(* CODESYS project Estação 3 - separating V2 (2022).project

Project tree, tasks and I/O mapping:
  Device : CPX-CEC-C1-V3, Festo AG & Co. KG, order no. 3473128, version 3.5.7.37
      unmapped channels: Rotary switch
    application Application
      libraries: Standard, * (System)
      task MainTask (cyclic, interval t#20ms, priority 20) calls PLC_PRG
      program PLC_PRG [ST]
      global variables GVL
      function ATUALIZAR_VALORES [ST]
      program pisca_pisca [ST]
      program modo_entrada [ST]
      program modo_saida [ST]
      program teste_comunicacao [ST]
    PLC_Diagnosis : PLC-Diagnosis, Festo AG & Co. KG, version 3.5.4.1
    CPX_System : CPX_System, Festo AG & Co. KG, order no. 3473128, version 1.258
      CEC_C1_V3 : CEC-C1-V3, Festo AG & Co. KG, order no. 3473128, version 1.258
          settings:  = 0;  = 234279157108224;  = 335718592;  = 65535;  = 16885952;  = 13959208;  = 1f5d13d5;  = 5
      _8DI_8DO : 8DI/8DO, Festo AG & Co. KG, order no. 526257, version 1.258
          settings:  = 0;  = 1;  = 1;  = 1;  = 1;  = 0;  = 1;  = 1;  = 0;  = 0;  = 0;  = 0;  = 0;  = 0;  = 0;  = 0;  = 0;  = 0;  = 0;  = 0;  = 0;  = 0;  = 0;  = 0;  = 0;  = 0;  = 0;  = 0;  = 0;  = 0;  = 0;  = 0;  = 0;  = 0;  = 0;  = 0;  = 0;  = 0;  = 0;  = 0;
             = 0;  = 0;  = 0;  = 0;  = 0;  = 0;  = 0;  = 0;  = 0;  = 0;  = 0;  = 0;  = 0;  = 0;  = 0;  = 0;  = 0;  = 0;  = 0;  = 0;  = 0;  = 0;  = 0;  = 0;  = 0;  = 0;  = 0;  = 0;  = 0;  = 0;  = 0;  = 0;  = 0;  = 0;  = 0;  = 0;  = 0;  = 0;  = 0;  = 0;
             = 576751027668385792;  = 'PI%i.0.0.1=1';  = 'PI%i.0.1.1=1';  = 'PI%i.0.2.1=1';  = 'PI%i.1.0.1=1';  = 'PI%i.1.1.1=0';  = 'PI%i.1.4.2=1';  = 'PI%i.1.6.2=1';  = 'PI%i.6.0.1=0';  = 'PI%i.6.1.1=0';  = 'PI%i.6.2.1=0';  = 'PI%i.6.3.1=0';  = 'PI%i.6.4.1=0';  = 'PI%i.6.5.1=0';  = 'PI%i.6.6.1=0';  = 'PI%i.6.7.1=0';  = dd379be8;  = 6
          unmapped channels: Input 0, Output 0
      _8DI_8DO_1 : 8DI/8DO, Festo AG & Co. KG, order no. 526257, version 1.258
          settings:  = 0;  = 1;  = 1;  = 1;  = 1;  = 0;  = 1;  = 1;  = 0;  = 0;  = 0;  = 0;  = 0;  = 0;  = 0;  = 0;  = 0;  = 0;  = 0;  = 0;  = 0;  = 0;  = 0;  = 0;  = 0;  = 0;  = 0;  = 0;  = 0;  = 0;  = 0;  = 0;  = 0;  = 0;  = 0;  = 0;  = 0;  = 0;  = 0;  = 0;
             = 0;  = 0;  = 0;  = 0;  = 0;  = 0;  = 0;  = 0;  = 0;  = 0;  = 0;  = 0;  = 0;  = 0;  = 0;  = 0;  = 0;  = 0;  = 0;  = 0;  = 0;  = 0;  = 0;  = 0;  = 0;  = 0;  = 0;  = 0;  = 0;  = 0;  = 0;  = 0;  = 0;  = 0;  = 0;  = 0;  = 0;  = 0;  = 0;  = 0;
             = 576751027668385792;  = 'PI%i.0.0.1=1';  = 'PI%i.0.1.1=1';  = 'PI%i.0.2.1=1';  = 'PI%i.1.0.1=1';  = 'PI%i.1.1.1=0';  = 'PI%i.1.4.2=1';  = 'PI%i.1.6.2=1';  = 'PI%i.6.0.1=0';  = 'PI%i.6.1.1=0';  = 'PI%i.6.2.1=0';  = 'PI%i.6.3.1=0';  = 'PI%i.6.4.1=0';  = 'PI%i.6.5.1=0';  = 'PI%i.6.6.1=0';  = 'PI%i.6.7.1=0';  = dd4a6df2;  = 6
          unmapped channels: Input 0, Output 0
    Ethernet : Ethernet, 3S - Smart Software Solutions GmbH, version 3.5.10.0
        settings: IPAddress = [192,168,0,1]; SubnetMask = [255,255,255,0]; GatewayAddress = [0,0,0,0]; MACAddress = [16#00,16#00,16#00,16#00,16#00,16#00]; SaveCommunicationSettings = FALSE
      ModbusTCP_Slave_Device : ModbusTCP Slave Device, 3S - Smart Software Solutions GmbH, version 3.5.10.0
          unmapped channels: Inputs, Outputs
*)

// Device/Application/GVL
	
{attribute 'qualified_only'}
VAR_GLOBAL
//Entradas
	//Sensores
	S_inicio 	AT %IX1.0 :BOOL; //Sensor de inicio da esteira
	S_meio 	 	AT %IX1.1 :BOOL; //Sensor do meio da esteira
	S_fim 		AT %IX1.2 :BOOL; //Sensor do fim da esteira
	S_dist		AT %IX1.3 :BOOL; //Sensor de distancia (sinal digital)
	S_inicio_2 	AT %IX1.4  :BOOL; //Sensor de inicio da esteira 2
	//  	AT %IX1.5  :BOOL; //
	S_fim_2 	AT %IX1.6  :BOOL; //Sensor do fim da esteira 2
	
	
	//IHM
	Start_btn 		AT	%IX2.0	:BOOL;  //Botão de start
	Stop_btn 		AT	%IX2.1	:BOOL;	//Botão de stop (NF)
	Chave 			AT	%IX2.2	:BOOL;	//Chave auto/manual
	Reset_btn 		AT	%IX2.3	:BOOL;	//Botão de reset
	I4_IHM			AT	%IX2.4	:BOOL;	//Bit de saída 4 da IHM
	I5_IHM			AT	%IX2.5	:BOOL;	//Bit de saída 5 da IHM
	I6_IHM 			AT	%IX2.6	:BOOL;	//Bit de saída 6 da IHM
	I7_IHM			AT	%IX2.7	:BOOL;	//Bit de saída 7 da IHM

//Saídas
	//Atuadorres 			
	Esteira_frente 	AT	%QX0.0	:BOOL;	//Mover a esteira 1 para frente
	Esteira_tras 	AT	%QX0.1	:BOOL;	//Mover a esteira 1 para tras
	Separador 	 	AT	%QX0.2	:BOOL;	//Atuar separador
	Stopper		 	AT	%QX0.3	:BOOL;	//Avança stopper
	Esteira_frente_2 AT	%QX0.4	:BOOL;	//Mover a esteira 2 para frente
	Esteira_tras_2	 AT	%QX0.5	:BOOL;	//Mover a esteira 2 para tras
	//				AT	%QX0.6	:BOOL;	
	//	     		AT	%QX0.7	:BOOL;	
	
	//IHM				
	Start_LED		AT	%QX1.0	:BOOL;	//LED do botão de start
	Reset_LED 		AT	%QX1.1	:BOOL;	//LED do botão de reset
	Q1_LED 			AT	%QX1.2	:BOOL;	//LED sinalizador Q1
	Q2_LED			AT	%QX1.3	:BOOL;	//LED sinalizador Q2
	Q4_IHM			AT	%QX1.4	:BOOL;	//Saída Q4 IHM
	Q5_IHM			AT	%QX1.5	:BOOL;	//Saída Q5 IHM
	Q6_IHM			AT	%QX1.6	:BOOL;	//Saída Q6 IHM
	Q7_IHM 			AT	%QX1.7	:BOOL;	//Saída Q7 IHM
	
//MODBUS bits
	//Entradas
	Mod_I_0_0 		AT %IX4.0 : BOOL; //Iniciar a estação 
	Mod_I_0_1	 	AT %IX4.1 : BOOL; //Parar a estação
	Mod_I_0_2 		AT %IX4.2 : BOOL; //Reiniciar a estação
	Mod_I_0_3 		AT %IX4.3 : BOOL; //Modo entrada
	Mod_I_0_4 		AT %IX4.4 : BOOL; ///Modo saída
	Mod_I_0_5 		AT %IX4.5 : BOOL; //Teste de resposta da estação - IN
	Mod_I_0_6 		AT %IX4.6 : BOOL;
	Mod_I_0_7 		AT %IX4.7 : BOOL;
	Mod_I_1_0 		AT %IX5.0 : BOOL;
	Mod_I_1_1 		AT %IX5.1 : BOOL;
	Mod_I_1_2 		AT %IX5.2 : BOOL;
	Mod_I_1_3 		AT %IX5.3 : BOOL;
	Mod_I_1_4 		AT %IX5.4 : BOOL;
	Mod_I_1_5	 	AT %IX5.5 : BOOL;
	Mod_I_1_6 		AT %IX5.6 : BOOL;
	Mod_I_1_7 		AT %IX5.7 : BOOL;
	
	//Saídas
	Mod_Q_0_0 		AT %QX2.0 : BOOL; //Estação iniciada 					
	Mod_Q_0_1	 	AT %QX2.1 : BOOL; //Estação parada 					
	Mod_Q_0_2 		AT %QX2.2 : BOOL; //Estação em processo			
	Mod_Q_0_3 		AT %QX2.3 : BOOL; //Estação em modo de entrada
	Mod_Q_0_4 		AT %QX2.4 : BOOL; //Estação em modo de saída
	Mod_Q_0_5 		AT %QX2.5 : BOOL; //Teste de resposta da estação - OUT	


//Variáveis de lógica
	principal: BOOL;
	parada : BOOL;
	passo1: BOOL;	
	passo2: BOOL;
	passo3: BOOL;
	passo4: BOOL;
	passo5: BOOL;
	passo6: BOOL;
	passo7: BOOL;
	passo8: BOOL;
	
	start: BOOL; //Start geral
	stop: BOOL;  //Stop geral
	reset: BOOL; //Reset geral
	key: BOOL; //key geral
	
	estacao_iniciada:  BOOL; //Flag para sinalizar que a estação está iniciada e pode receber algum comando
	estacao_parada: BOOL;	//Flag que sinaliza estação parada
	estacao_em_processo: BOOL; //Flag que sinaliza a estação em processo
	ligar_pisca: BOOL := FALSE; //Flag para ligar e desligar o pisca pisca
	modo_entrada: BOOL; //Quando setado, a estação entra em modo de saída de peças
	modo_saida: BOOL; //Quando setado, a estação entra em modo de entrada de peças
	Peca_robo: BOOL; //Quando for TRUE, a peça irá para a montagem no robô, se for FALSE irá para a montatgem da tampinha

END_VAR

// Device/Application/PLC_PRG
PROGRAM PLC_PRG
VAR
	TONInst4: Ton;
	TON_4: BOOL;
	TON_3: BOOL;
	TONInst3: Ton;
	TONInst1: Ton;
	TON_1: BOOL;
	TONInst2: Ton;
	TON_2: BOOL;
	TONInst5: Ton;
	TON_5: BOOL;
END_VAR

modo_entrada();
modo_saida();
pisca_pisca();
teste_comunicacao();
ATUALIZAR_VALORES();

END_PROGRAM

// Device/Application/modo_entrada
PROGRAM modo_entrada
VAR

	TON_temp_1: TON;
	TON_1: BOOL;
	
	TON_temp_2: TON;
	TON_2: BOOL;	
	
	PASSOS: INT;
	
END_VAR

TON_temp_1(IN := TON_1, PT:= T#0.5S);
TON_temp_2(IN := TON_2, PT:= T#0.4S);

IF NOT gvl.estacao_parada AND gvl.estacao_iniciada THEN
	
	IF (gvl.modo_entrada AND NOT gvl.modo_saida AND PASSOS = 0) THEN
		GVL.Q4_IHM := TRUE;
	END_IF
	
	IF ((gvl.modo_entrada AND NOT gvl.modo_saida) OR PASSOS = 1) AND gvl.S_inicio THEN
		GVL.Q4_IHM := FALSE;
		gvl.ligar_pisca := TRUE;
		gvl.estacao_em_processo := TRUE;
		gvl.Stopper := FALSE;	
		gvl.Esteira_frente := TRUE;
		gvl.Esteira_frente_2 := TRUE;
		gvl.Separador := TRUE;
		PASSOS := 1;
	END_IF
	
	
	IF PASSOS = 1 AND NOT gvl.S_fim_2 THEN
		TON_1 := TRUE;
	END_IF
	
	IF TON_temp_1.Q THEN
		TON_1 := FALSE;
		gvl.ligar_pisca := FALSE;
		gvl.estacao_em_processo := FALSE;
		PASSOS := 0;
		gvl.Esteira_frente := FALSE;
		gvl.Esteira_frente_2 := FALSE;
		gvl.Separador := FALSE;
	END_IF
	
	ELSE
		gvl.Esteira_frente := FALSE;
		gvl.Esteira_frente_2 := FALSE;
	
END_IF

END_PROGRAM

// Device/Application/modo_saida
PROGRAM modo_saida
VAR
	
	TON_temp_1: TON;
	TON_1: BOOL;
	
	TON_temp_2: TON;
	TON_2: BOOL;	
	
	PASSOS: INT;	

END_VAR

TON_temp_1(IN := TON_1, PT:= T#5S);
TON_temp_2(IN := TON_2, PT:= T#0.4S);

IF NOT gvl.estacao_parada AND gvl.estacao_iniciada THEN
	
	IF ((NOT gvl.modo_entrada AND gvl.modo_saida) OR PASSOS = 1) AND NOT  gvl.S_fim_2 THEN
		gvl.ligar_pisca := TRUE;
		gvl.estacao_em_processo := TRUE;
		gvl.Stopper := TRUE;	
		gvl.Esteira_frente := TRUE;
		gvl.Esteira_tras_2 := TRUE;
		gvl.Separador := FALSE;
		TON_1 := FALSE;
		PASSOS := 1;
	END_IF
	
	
	IF PASSOS = 1 AND NOT gvl.S_fim THEN
		TON_1 := TRUE;
	END_IF
	
	IF TON_temp_1.Q THEN
		TON_1 := FALSE;
		gvl.estacao_em_processo := FALSE;
		gvl.Stopper := FALSE;
		gvl.ligar_pisca := FALSE;
		PASSOS := 0;
		gvl.Esteira_frente := FALSE;
		gvl.Esteira_tras_2 := FALSE;
		gvl.Separador := FALSE;
	END_IF
	
	ELSE
		gvl.Esteira_frente := FALSE;
		gvl.Esteira_tras_2 := FALSE;
END_IF

END_PROGRAM

// Device/Application/pisca_pisca
PROGRAM pisca_pisca
VAR
	
	TON_temp_1: TON;
	TON_1: BOOL;
	TON_temp_2: TON;
	TON_2: BOOL;
	
	passo: INT;
END_VAR

TON_temp_1(IN := TON_1, PT:= T#0.2S);
TON_temp_2(IN := TON_2, PT:= T#0.2S);

IF gvl.ligar_pisca AND (passo = 0)  THEN
	TON_1 := TRUE;
	passo := 1;
END_IF

IF NOT gvl.ligar_pisca THEN
	TON_1 := FALSE;
	TON_2 := FALSE;
	GVL.Q2_LED := FALSE;
	passo := 0;
END_IF

IF TON_temp_1.Q THEN
	TON_1 := FALSE;
	TON_2 := TRUE;
	GVL.Q2_LED := TRUE;
END_IF

IF TON_temp_2.Q THEN
	TON_1 := TRUE;
	TON_2 := FALSE;
	GVL.Q2_LED := FALSE;
END_IF

END_PROGRAM

// Device/Application/teste_comunicacao
PROGRAM teste_comunicacao
VAR
	
	TON_temp_1: TON;
	TON_1: BOOL;	

END_VAR

gvl.Mod_Q_0_5 := gvl.Mod_I_0_5;

END_PROGRAM

// Device/Application/ATUALIZAR_VALORES
FUNCTION ATUALIZAR_VALORES : INT
VAR
END_VAR

GVL.Mod_Q_0_0 := GVL.estacao_iniciada;
GVL.Mod_Q_0_1 := GVL.estacao_parada;
GVL.Mod_Q_0_2 := GVL.estacao_em_processo;
GVL.Mod_Q_0_3 := GVL.modo_entrada;
GVL.Mod_Q_0_4 := GVL.modo_saida;

gvl.modo_entrada := GVL.Mod_I_0_3; //Seta modo de entrada
gvl.modo_saida 	 := GVL.Mod_I_0_4; //Seta modo de saída

GVL.Mod_Q_0_3 := GVL.modo_entrada;
GVL.Mod_Q_0_4 := GVL.modo_saida;


IF GVL.Start_btn OR GVL.Mod_I_0_0 THEN  //Atualização do valor da variável de start
	GVL.start := TRUE;
	IF NOT gvl.estacao_parada THEN
		GVL.estacao_iniciada := TRUE;
		GVL.Q1_LED := TRUE;
	END_IF
	ELSE
	GVL.start := FALSE;
END_IF

IF NOT GVL.Stop_btn OR GVL.Mod_I_0_1 THEN //Atualização do valor da variável de stop
	GVL.stop := TRUE;
	GVL.estacao_iniciada := FALSE;
	gvl.estacao_parada := TRUE;
	GVL.Q1_LED := FALSE;
	gvl.estacao_em_processo := FALSE;
	gvl.ligar_pisca := FALSE;
	ELSE
	GVL.stop := FALSE;
END_IF

IF GVL.Reset_btn OR GVL.Mod_I_0_2 THEN //Atualização do valor da variável de reset
	GVL.reset := TRUE;
	gvl.estacao_parada := FALSE;
	gvl.modo_entrada := FALSE;
	gvl.modo_saida := FALSE;
	gvl.Separador := FALSE;
	ELSE
	GVL.reset := FALSE;	
END_IF

IF GVL.Chave OR GVL.Mod_I_0_3 THEN //Atualização do valor da variável da chave
	GVL.key := TRUE;
	ELSE
	GVL.key := FALSE;
END_IF

END_FUNCTION
